// Function block used for physical output control
FUNCTION_BLOCK FB_Output IMPLEMENTS I_Output
VAR_INPUT

END_VAR
VAR_OUTPUT

END_VAR
VAR
	bOut	AT %Q*	:	BOOL;	// Physical output
	sDescription	:	STRING;	// Description of the output
	bOutAuto		:	BOOL;	// This value will be used in automatic mode
	bManualMode		:	BOOL;	// Turns on and off manual mode
	bOutManual		:	BOOL;	// This value will be used in manual mode
END_VAR

{attribute 'monitoring' := 'variable'}
PROPERTY Description : STRING
GET
Description := sDescription;
END_GET
SET
sDescription := Description;
END_SET
END_PROPERTY

{attribute 'monitoring' := 'variable'}
PROPERTY ManualMode : BOOL
GET
ManualMode := bManualMode;
END_GET
SET
bManualMode := ManualMode;
END_SET
END_PROPERTY

{attribute 'monitoring' := 'variable'}
PROPERTY OutAuto : BOOL
GET
OutAuto := bOut;
END_GET
SET
bOutAuto := OutAuto;
IF NOT bManualMode THEN
	bOut := bOutAuto;
END_IF
END_SET
END_PROPERTY

{attribute 'monitoring' := 'variable'}
PROPERTY OutManual : BOOL
GET
OutManual := bOut;
END_GET
SET
bOutManual := OutManual;
IF bManualMode THEN
	bOut := bOutManual;
END_IF
END_SET
END_PROPERTY

END_FUNCTION_BLOCK

(* stored: Version 1.1.0.1, ProductVersion 3.1.4024.12
   POU FB_Output: Id {5cc7aa47-0b26-4ec9-a125-9e3eeb4b5f3f}, SpecialFunc None
   Property Description: Id {90955d4d-0c81-49ef-87f5-27aae1123746}
   Get Get: Id {255e2ff7-f769-4b1e-a72c-be7053c3b03f}
   Set Set: Id {135f6c88-e1fc-4837-acc7-af66d6b4b92c}
   Property ManualMode: Id {7786d54d-55ec-4d6c-8e82-a6dc55804da9}
   Get Get: Id {476b28a4-3c83-4afb-946a-fc076eeb90fd}
   Set Set: Id {919cd098-c48a-46ea-9ef2-6a845ac35a19}
   Property OutAuto: Id {982a39c5-a113-4ab1-874f-5eee41d6a309}
   Get Get: Id {c6945c41-bd22-4b4e-96fb-077a6d8f8e57}
   Set Set: Id {e761d01d-b198-498b-a072-a04074410495}
   Property OutManual: Id {9e156cd2-fbe0-4f81-a7bc-ea8f8c990eb9}
   Get Get: Id {873ae1ac-e1f3-4f11-b18c-a54d3bc1f333}
   Set Set: Id {044bd78b-aa8c-4c36-9f93-f0cf201a8b69} *)
